TYPE EL3356 :
STRUCT
	ch1		:DINT;
END_STRUCT
END_TYPE

(* stored: Version 1.1.0.1, ProductVersion 3.1.4024.12
   DUT EL3356: Id {3dae1f61-6168-43fa-8c81-6963105ffd58} *)
